FUNCTION_BLOCK BfbIntersectionMutex
  (* Standard: 61499-2 *)
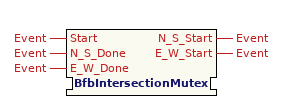
  EVENT_INPUT
    Start;
    N_S_Done;
    E_W_Done;
  END_EVENT
  EVENT_OUTPUT
    N_S_Start;
    E_W_Start;
  END_EVENT
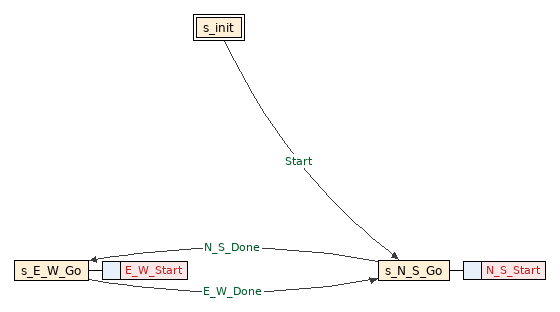
  EC_STATES
    s_init;
    s_N_S_Go : -> N_S_Start;
    s_E_W_Go : -> E_W_Start;
  END_STATES
  EC_TRANSITIONS
    s_init TO s_N_S_Go := Start;
    s_N_S_Go TO s_E_W_Go := N_S_Done;
    s_E_W_Go TO s_N_S_Go := E_W_Done;
  END_TRANSITIONS
END_FUNCTION_BLOCK
